{attribute 'qualified_only'}
VAR_GLOBAL
		Device_1_EtherCAT : Device_1_EtherCAT_9EEE92A7;
END_VAR

(* stored: Version 1.2.0.0, ProductVersion 3.1.4024.9
   GVL GVL_iXlinker: Id {e50bb25e-dbe3-43df-8564-f2542ac71179} *)
